// TIA Portal V18 export
TYPE "UDT_Store_OpMode"
// stored: IsFailsafeCompliant false
   STRUCT
      cPreviousOne { S7_SetPoint := 'True'} : Byte;
      cActual { S7_SetPoint := 'True'} : Byte;   // Поточний/Актуальний режим роботи
      cTarget { S7_SetPoint := 'True'} : Byte;   // Вибраний режим роботи, але ще не дійшли до нього
      cPreselectedOpMode : Byte;   // 0-Protection/1-economy/2-PreComfort/3-Comfort/4-Auto
   END_STRUCT;
END_TYPE
